// TIA Portal V19 export
DATA_BLOCK "instReadCanProcessImage"   // DB5
// stored: AutoNumber false, InstanceOfName ReadCanProcessImage, InstanceOfType FB
"ReadCanProcessImage"
   // VAR_OUTPUT
   //    Busy : Bool;
   //    Error : Bool;
   //    Len : UInt;
   //    Status : DWord;
   //    Valid : Bool;
   // END_VAR
   // VAR_IN_OUT
   //    CanProcessImage : Array[0..31] of Byte;
   // END_VAR
BEGIN
END_DATA_BLOCK
